// Mitsubishi GX Works2 project: InterLock_SelfHolding2   PLC: Q03UDV

PROGRAM MAIN
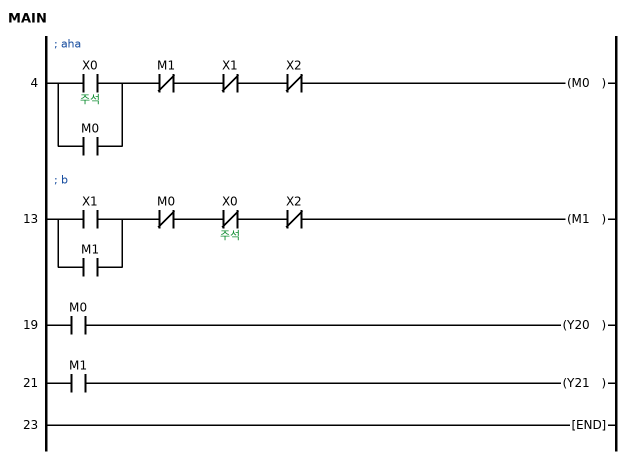
; aha
4     LD      X0  ; 주석
      OR      M0
      ANI     M1
      ANI     X1
      ANI     X2
      OUT     M0
; b
13    LD      X1
      OR      M1
      ANI     M0
      ANI     X0  ; 주석
      ANI     X2
      OUT     M1
19    LD      M0
      OUT     Y20
21    LD      M1
      OUT     Y21
23    END
END_PROGRAM
